Fanuc KAREL source: IO0119.KL

PROGRAM IO0119
%STACKSIZE=65535
%PRIORITY=65535
%NOLOCKGROUP
ROUTINE RTEST FROM IO0119
ROUTINE RTEST
VAR
L1 : ARRAY[3] OF INTEGER
L2 : XYZWPR
L3 : JOINTPOS9
L4 : POSITION
S1 : INTEGER
U2C_38 : REAL -- ASSUMED 2C source type; see uncertainty report
U2C_39 : REAL -- ASSUMED 2C source type; see uncertainty report
U2C_40 : BOOLEAN -- ASSUMED 2C source type; see uncertainty report
U2C_41 : INTEGER -- ASSUMED 2C source type; see uncertainty report
BEGIN
S1=1
L1[1]=2
U2C_40=TRUE
U2C_41=1065353216
-- UNSAFE_SOURCE_IR line 19: IF (native_io_value(9, (S1 + 1)) = 1) THEN
S1=(S1 + 1)
ENDIF
END RTEST
BEGIN
RTEST
END IO0119
